% RSLogix 500 project BLUE BANNER_ORGANIC_DUMP_APR_09_2021_FAST_SLOW_BOTH_BAK083.RSS, saved by version 11.00.00.00 %
PROJECT "CCHDUMP"    % processor: MicroLogix 1400 %

PROGRAM FILES
  LAD 2   72 rungs

DATA FILES
  O0 OUTPUT  7 elements
  I1 INPUT  9 elements
  S2 STATUS  66 elements
  B3 BINARY  4 elements
  T4 TIMER  20 elements
  C5 COUNTER  1 elements
  R6 CONTROL  1 elements
  N7 INTEGER  1 elements
  F8 FLOAT  4 elements

LADDER 2
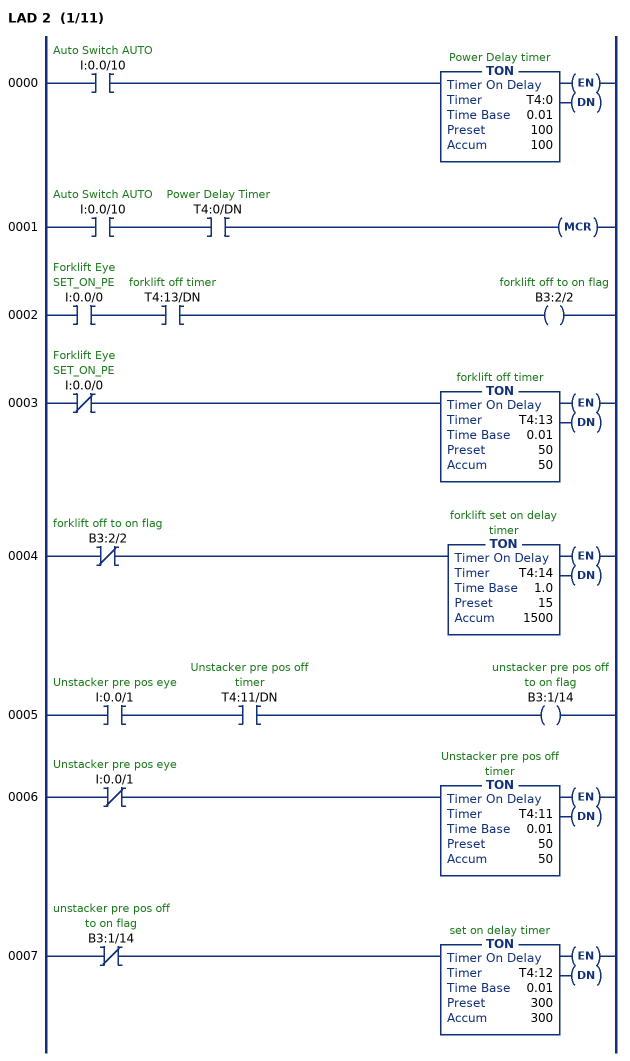
% Rung: 0 %
SOR XIC I:0.0/10 TON T4:0 0.01 100 100 EOR
%   I:0.0/10  AUTO  "Auto Switch" %
%   T4:0  "Power Delay timer" %
% Rung: 1 %
SOR XIC I:0.0/10 XIC T4:0/DN MCR EOR
%   I:0.0/10  AUTO  "Auto Switch" %
%   T4:0/DN  "Power Delay Timer" %
% Rung: 2 %
SOR XIC I:0.0/0 XIC T4:13/DN OTE B3:2/2 EOR
%   I:0.0/0  SET_ON_PE  "Forklift Eye" %
%   T4:13  "forklift off timer" %
%   B3:2/2  "forklift off to on flag" %
% Rung: 3 %
SOR XIO I:0.0/0 TON T4:13 0.01 50 50 EOR
%   I:0.0/0  SET_ON_PE  "Forklift Eye" %
%   T4:13  "forklift off timer" %
% Rung: 4 %
SOR XIO B3:2/2 TON T4:14 1.0 15 1500 EOR
%   B3:2/2  "forklift off to on flag" %
%   T4:14  "forklift set on delay timer" %
% Rung: 5 %
SOR XIC I:0.0/1 XIC T4:11/DN OTE B3:1/14 EOR
%   I:0.0/1  "Unstacker pre pos eye" %
%   T4:11  "Unstacker pre pos off timer" %
%   B3:1/14  "unstacker pre pos off to on flag" %
% Rung: 6 %
SOR XIO I:0.0/1 TON T4:11 0.01 50 50 EOR
%   I:0.0/1  "Unstacker pre pos eye" %
%   T4:11  "Unstacker pre pos off timer" %
% Rung: 7 %
SOR XIO B3:1/14 TON T4:12 0.01 300 300 EOR
%   B3:1/14  "unstacker pre pos off to on flag" %
%   T4:12  "set on delay timer" %

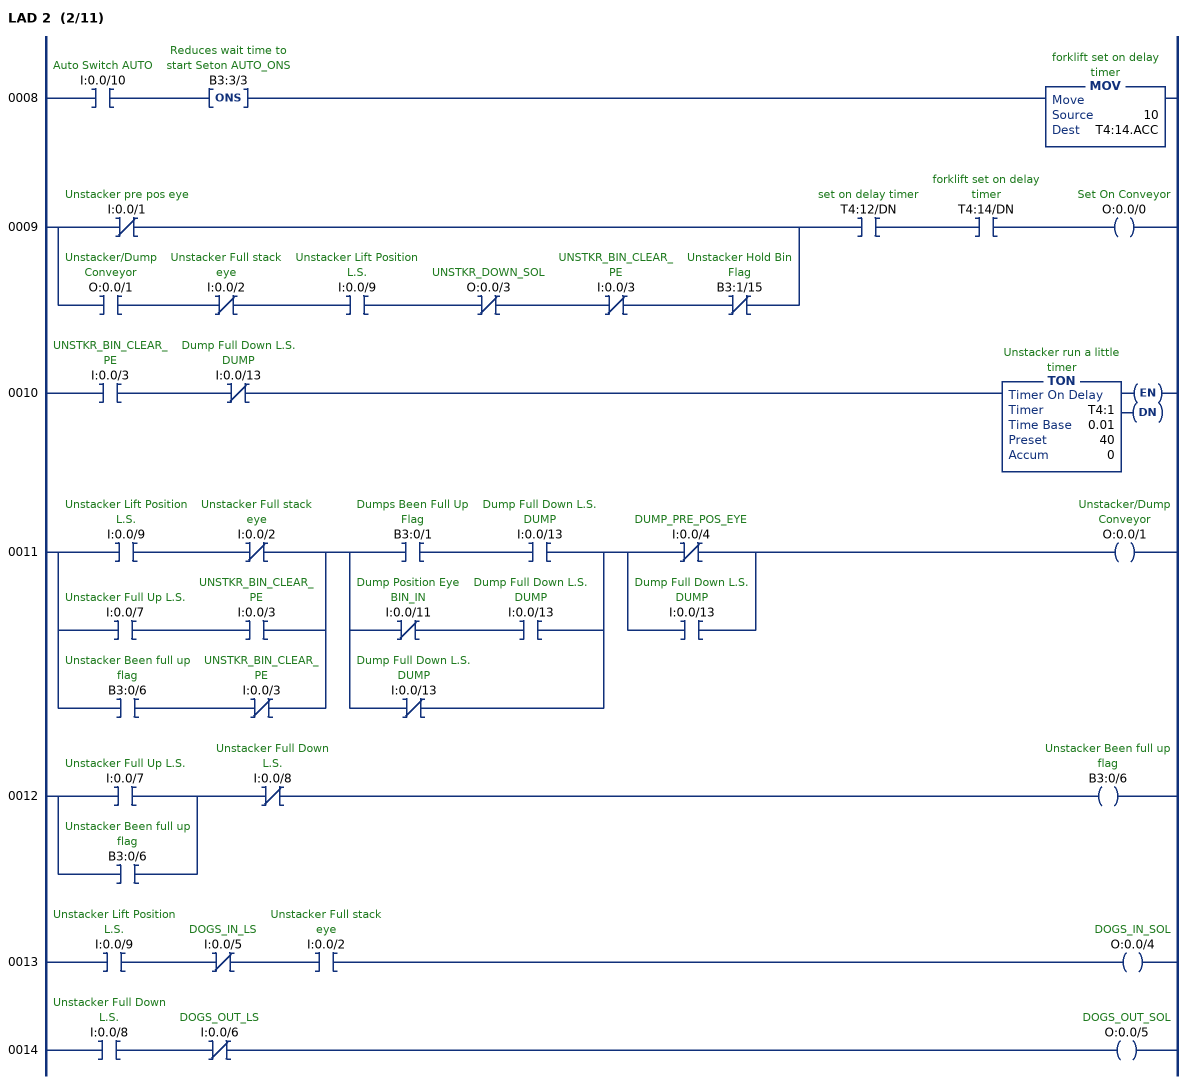
% Rung: 8 %
SOR XIC I:0.0/10 ONS B3:3/3 MOV 10 T4:14.ACC EOR
%   I:0.0/10  AUTO  "Auto Switch" %
%   B3:3/3  AUTO_ONS  "Reduces wait time to start Seton" %
%   T4:14  "forklift set on delay timer" %
% Rung: 9 %
SOR BST XIO I:0.0/1 NXB XIC O:0.0/1 XIO I:0.0/2 XIC I:0.0/9 XIO O:0.0/3 XIO I:0.0/3 XIO B3:1/15 BND XIC T4:12/DN XIC T4:14/DN OTE O:0.0/0 EOR
%   I:0.0/1  "Unstacker pre pos eye" %
%   O:0.0/1  "Unstacker/Dump Conveyor" %
%   I:0.0/2  "Unstacker Full stack eye" %
%   I:0.0/9  "Unstacker Lift Position L.S." %
%   O:0.0/3  UNSTKR_DOWN_SOL %
%   I:0.0/3  UNSTKR_BIN_CLEAR_PE %
%   B3:1/15  "Unstacker Hold Bin Flag" %
%   T4:12  "set on delay timer" %
%   T4:14  "forklift set on delay timer" %
%   O:0.0/0  "Set On Conveyor" %
% Rung: 10 %
SOR XIC I:0.0/3 XIO I:0.0/13 TON T4:1 0.01 40 0 EOR
%   I:0.0/3  UNSTKR_BIN_CLEAR_PE %
%   I:0.0/13  DUMP  "Dump Full Down L.S." %
%   T4:1  "Unstacker run a little timer" %
% Rung: 11 %
SOR BST XIC I:0.0/9 XIO I:0.0/2 NXB XIC I:0.0/7 XIC I:0.0/3 NXB XIC B3:0/6 XIO I:0.0/3 BND BST XIC B3:0/1 XIC I:0.0/13 NXB XIO I:0.0/11 XIC I:0.0/13 NXB XIO I:0.0/13 BND BST XIO I:0.0/4 NXB XIC I:0.0/13 BND OTE O:0.0/1 EOR
%   I:0.0/9  "Unstacker Lift Position L.S." %
%   I:0.0/2  "Unstacker Full stack eye" %
%   I:0.0/7  "Unstacker Full Up L.S." %
%   I:0.0/3  UNSTKR_BIN_CLEAR_PE %
%   B3:0/6  "Unstacker Been full up flag" %
%   B3:0/1  "Dumps Been Full Up Flag" %
%   I:0.0/13  DUMP  "Dump Full Down L.S." %
%   I:0.0/11  BIN_IN  "Dump Position Eye" %
%   I:0.0/4  DUMP_PRE_POS_EYE %
%   O:0.0/1  "Unstacker/Dump Conveyor" %
% Rung: 12 %
SOR BST XIC I:0.0/7 NXB XIC B3:0/6 BND XIO I:0.0/8 OTE B3:0/6 EOR
%   I:0.0/7  "Unstacker Full Up L.S." %
%   B3:0/6  "Unstacker Been full up flag" %
%   I:0.0/8  "Unstacker Full Down L.S." %
% Rung: 13 %
SOR XIC I:0.0/9 XIO I:0.0/5 XIC I:0.0/2 OTE O:0.0/4 EOR
%   I:0.0/9  "Unstacker Lift Position L.S." %
%   I:0.0/5  DOGS_IN_LS %
%   I:0.0/2  "Unstacker Full stack eye" %
%   O:0.0/4  DOGS_IN_SOL %
% Rung: 14 %
SOR XIC I:0.0/8 XIO I:0.0/6 OTE O:0.0/5 EOR
%   I:0.0/8  "Unstacker Full Down L.S." %
%   I:0.0/6  DOGS_OUT_LS %
%   O:0.0/5  DOGS_OUT_SOL %

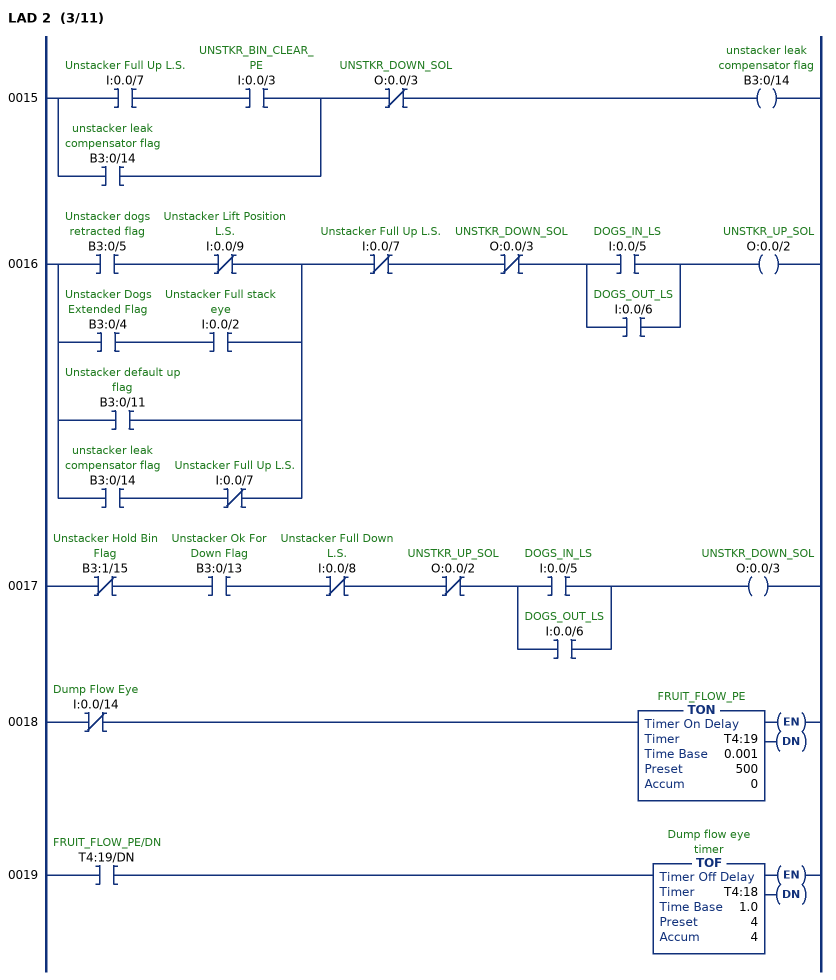
% Rung: 15 %
SOR BST XIC I:0.0/7 XIC I:0.0/3 NXB XIC B3:0/14 BND XIO O:0.0/3 OTE B3:0/14 EOR
%   I:0.0/7  "Unstacker Full Up L.S." %
%   I:0.0/3  UNSTKR_BIN_CLEAR_PE %
%   B3:0/14  "unstacker leak compensator flag" %
%   O:0.0/3  UNSTKR_DOWN_SOL %
% Rung: 16 %
SOR BST XIC B3:0/5 XIO I:0.0/9 NXB XIC B3:0/4 XIC I:0.0/2 NXB XIC B3:0/11 NXB XIC B3:0/14 XIO I:0.0/7 BND XIO I:0.0/7 XIO O:0.0/3 BST XIC I:0.0/5 NXB XIC I:0.0/6 BND OTE O:0.0/2 EOR
%   B3:0/5  "Unstacker dogs retracted flag" %
%   I:0.0/9  "Unstacker Lift Position L.S." %
%   B3:0/4  "Unstacker Dogs Extended Flag" %
%   I:0.0/2  "Unstacker Full stack eye" %
%   B3:0/11  "Unstacker default up flag" %
%   B3:0/14  "unstacker leak compensator flag" %
%   I:0.0/7  "Unstacker Full Up L.S." %
%   O:0.0/3  UNSTKR_DOWN_SOL %
%   I:0.0/5  DOGS_IN_LS %
%   I:0.0/6  DOGS_OUT_LS %
%   O:0.0/2  UNSTKR_UP_SOL %
% Rung: 17 %
SOR XIO B3:1/15 XIC B3:0/13 XIO I:0.0/8 XIO O:0.0/2 BST XIC I:0.0/5 NXB XIC I:0.0/6 BND OTE O:0.0/3 EOR
%   B3:1/15  "Unstacker Hold Bin Flag" %
%   B3:0/13  "Unstacker Ok For Down Flag" %
%   I:0.0/8  "Unstacker Full Down L.S." %
%   O:0.0/2  UNSTKR_UP_SOL %
%   I:0.0/5  DOGS_IN_LS %
%   I:0.0/6  DOGS_OUT_LS %
%   O:0.0/3  UNSTKR_DOWN_SOL %
% Rung: 18 %
SOR XIO I:0.0/14 TON T4:19 0.001 500 0 EOR
%   I:0.0/14  "Dump Flow Eye" %
%   T4:19  FRUIT_FLOW_PE %
% Rung: 19 %
SOR XIC T4:19/DN TOF T4:18 1.0 4 4 EOR
%   T4:19  FRUIT_FLOW_PE %
%   T4:18  "Dump flow eye timer" %

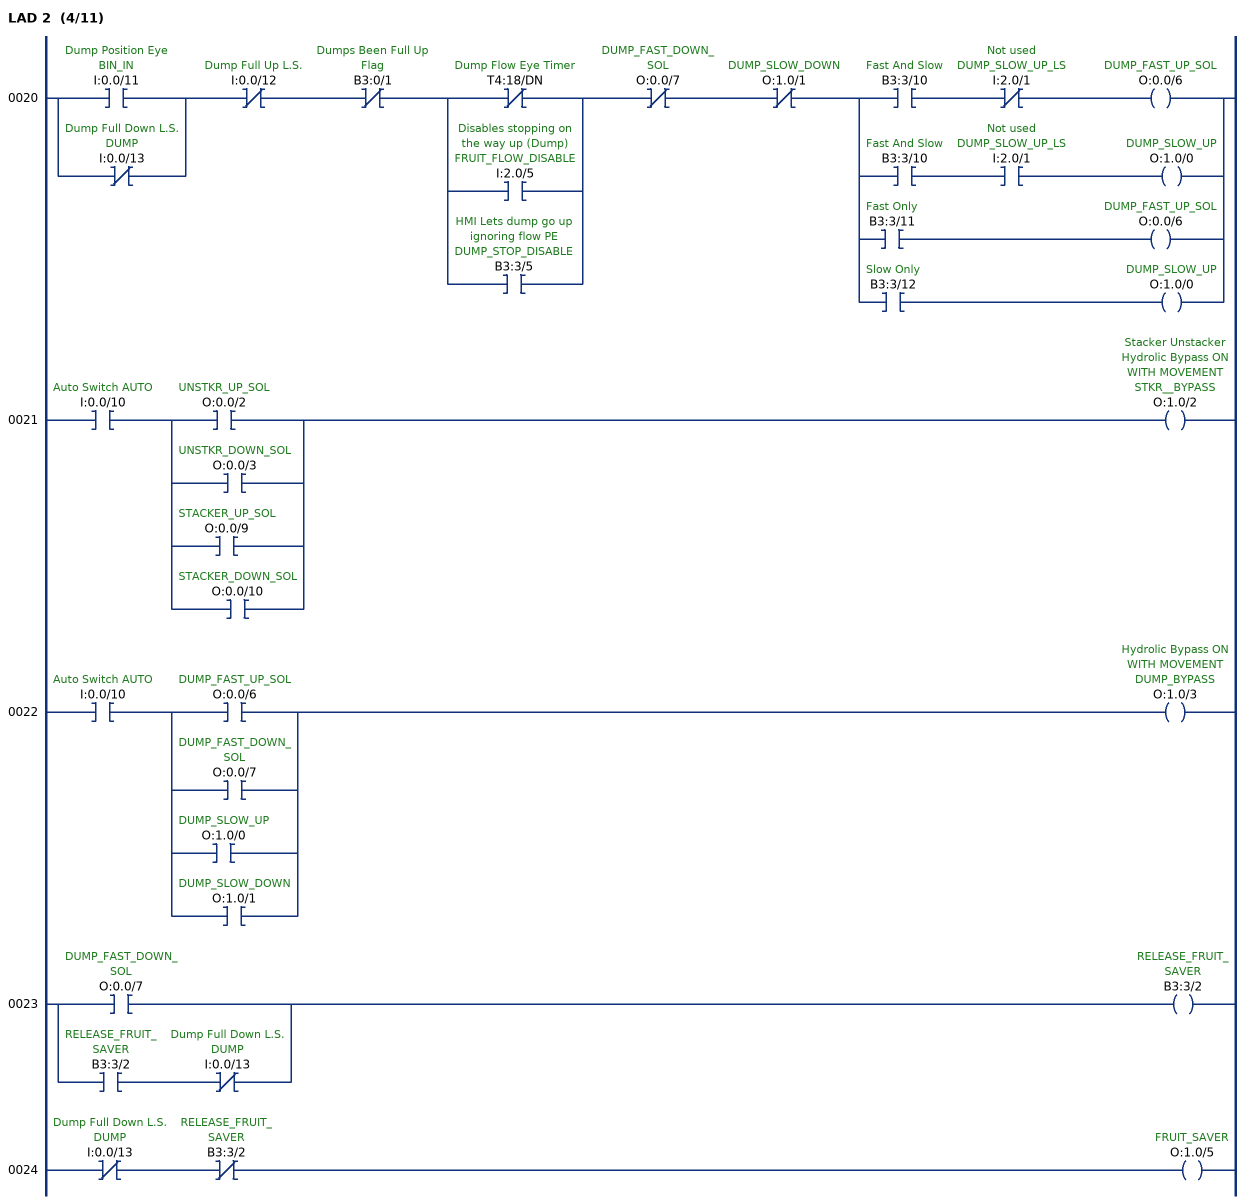
% Rung: 20 %
SOR BST XIC I:0.0/11 NXB XIO I:0.0/13 BND XIO I:0.0/12 XIO B3:0/1 BST XIO T4:18/DN NXB BST XIC I:2.0/5 NXB XIC B3:3/5 BND BND XIO O:0.0/7 XIO O:1.0/1 BST XIC B3:3/10 XIO I:2.0/1 OTE O:0.0/6 NXB XIC B3:3/10 XIC I:2.0/1 OTE O:1.0/0 NXB XIC B3:3/11 OTE O:0.0/6 NXB XIC B3:3/12 OTE O:1.0/0 BND EOR
%   I:0.0/11  BIN_IN  "Dump Position Eye" %
%   I:0.0/13  DUMP  "Dump Full Down L.S." %
%   I:0.0/12  "Dump Full Up L.S." %
%   B3:0/1  "Dumps Been Full Up Flag" %
%   T4:18/DN  "Dump Flow Eye Timer" %
%   I:2.0/5  FRUIT_FLOW_DISABLE  "Disables stopping on the way up (Dump)" %
%   B3:3/5  DUMP_STOP_DISABLE  "HMI Lets dump go up ignoring flow PE" %
%   O:0.0/7  DUMP_FAST_DOWN_SOL %
%   O:1.0/1  DUMP_SLOW_DOWN %
%   B3:3/10  "Fast And Slow" %
%   I:2.0/1  DUMP_SLOW_UP_LS  "Not used" %
%   O:0.0/6  DUMP_FAST_UP_SOL %
%   O:1.0/0  DUMP_SLOW_UP %
%   B3:3/11  "Fast Only" %
%   B3:3/12  "Slow Only" %
% Rung: 21 %
SOR XIC I:0.0/10 BST XIC O:0.0/2 NXB BST XIC O:0.0/3 NXB BST XIC O:0.0/9 NXB XIC O:0.0/10 BND BND BND OTE O:1.0/2 EOR
%   I:0.0/10  AUTO  "Auto Switch" %
%   O:0.0/2  UNSTKR_UP_SOL %
%   O:0.0/3  UNSTKR_DOWN_SOL %
%   O:0.0/9  STACKER_UP_SOL %
%   O:0.0/10  STACKER_DOWN_SOL %
%   O:1.0/2  STKR__BYPASS  "Stacker Unstacker Hydrolic Bypass ON WITH MOVEMENT" %
% Rung: 22 %
SOR XIC I:0.0/10 BST XIC O:0.0/6 NXB BST XIC O:0.0/7 NXB BST XIC O:1.0/0 NXB XIC O:1.0/1 BND BND BND OTE O:1.0/3 EOR
%   I:0.0/10  AUTO  "Auto Switch" %
%   O:0.0/6  DUMP_FAST_UP_SOL %
%   O:0.0/7  DUMP_FAST_DOWN_SOL %
%   O:1.0/0  DUMP_SLOW_UP %
%   O:1.0/1  DUMP_SLOW_DOWN %
%   O:1.0/3  DUMP_BYPASS  "Hydrolic Bypass ON WITH MOVEMENT" %
% Rung: 23 %
SOR BST XIC O:0.0/7 NXB XIC B3:3/2 XIO I:0.0/13 BND OTE B3:3/2 EOR
%   O:0.0/7  DUMP_FAST_DOWN_SOL %
%   B3:3/2  RELEASE_FRUIT_SAVER %
%   I:0.0/13  DUMP  "Dump Full Down L.S." %
% Rung: 24 %
SOR XIO I:0.0/13 XIO B3:3/2 OTE O:1.0/5 EOR
%   I:0.0/13  DUMP  "Dump Full Down L.S." %
%   B3:3/2  RELEASE_FRUIT_SAVER %
%   O:1.0/5  FRUIT_SAVER %

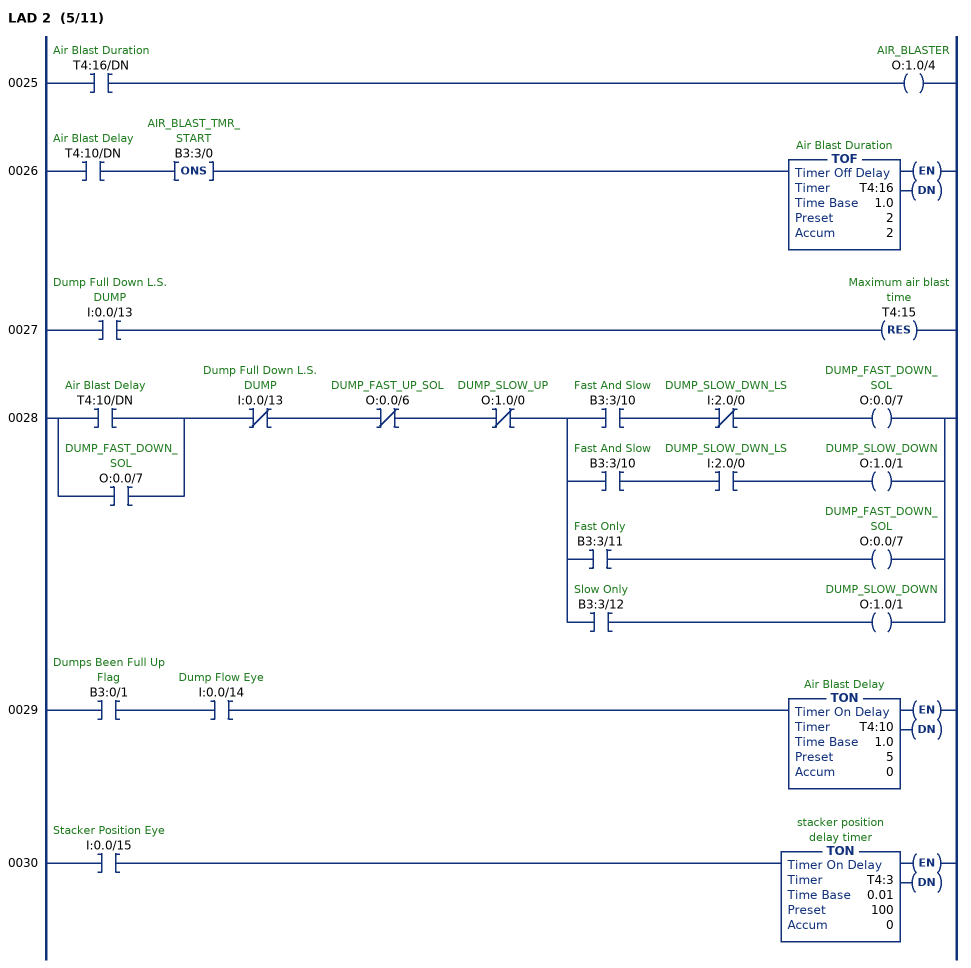
% Rung: 25 %
SOR XIC T4:16/DN OTE O:1.0/4 EOR
%   T4:16  "Air Blast Duration" %
%   O:1.0/4  AIR_BLASTER %
% Rung: 26 %
SOR XIC T4:10/DN ONS B3:3/0 TOF T4:16 1.0 2 2 EOR
%   T4:10  "Air Blast Delay" %
%   B3:3/0  AIR_BLAST_TMR_START %
%   T4:16  "Air Blast Duration" %
% Rung: 27 %
SOR XIC I:0.0/13 RES T4:15 EOR
%   I:0.0/13  DUMP  "Dump Full Down L.S." %
%   T4:15  "Maximum air blast time" %
% Rung: 28 %
SOR BST XIC T4:10/DN NXB XIC O:0.0/7 BND XIO I:0.0/13 XIO O:0.0/6 XIO O:1.0/0 BST XIC B3:3/10 XIO I:2.0/0 OTE O:0.0/7 NXB XIC B3:3/10 XIC I:2.0/0 OTE O:1.0/1 NXB XIC B3:3/11 OTE O:0.0/7 NXB XIC B3:3/12 OTE O:1.0/1 BND EOR
%   T4:10  "Air Blast Delay" %
%   O:0.0/7  DUMP_FAST_DOWN_SOL %
%   I:0.0/13  DUMP  "Dump Full Down L.S." %
%   O:0.0/6  DUMP_FAST_UP_SOL %
%   O:1.0/0  DUMP_SLOW_UP %
%   B3:3/10  "Fast And Slow" %
%   I:2.0/0  DUMP_SLOW_DWN_LS %
%   O:1.0/1  DUMP_SLOW_DOWN %
%   B3:3/11  "Fast Only" %
%   B3:3/12  "Slow Only" %
% Rung: 29 %
SOR XIC B3:0/1 XIC I:0.0/14 TON T4:10 1.0 5 0 EOR
%   B3:0/1  "Dumps Been Full Up Flag" %
%   I:0.0/14  "Dump Flow Eye" %
%   T4:10  "Air Blast Delay" %
% Rung: 30 %
SOR XIC I:0.0/15 TON T4:3 0.01 100 0 EOR
%   I:0.0/15  "Stacker Position Eye" %
%   T4:3  "stacker position delay timer" %

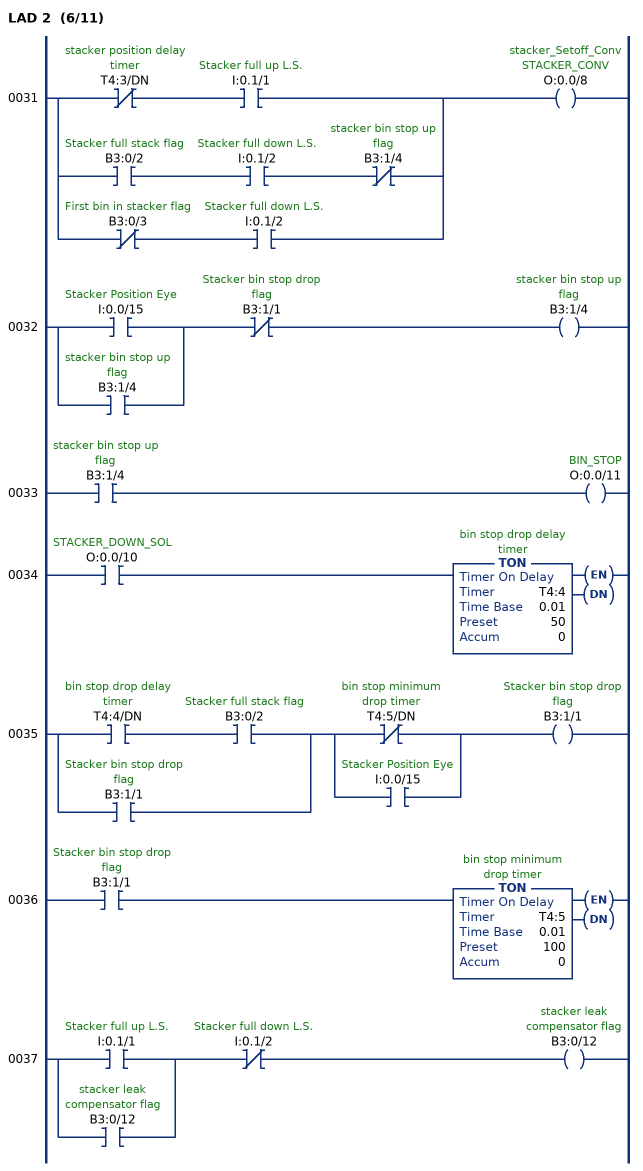
% Rung: 31 %
SOR BST XIO T4:3/DN XIC I:0.1/1 NXB XIC B3:0/2 XIC I:0.1/2 XIO B3:1/4 NXB XIO B3:0/3 XIC I:0.1/2 BND OTE O:0.0/8 EOR
%   T4:3  "stacker position delay timer" %
%   I:0.1/1  "Stacker full up L.S." %
%   B3:0/2  "Stacker full stack flag" %
%   I:0.1/2  "Stacker full down L.S." %
%   B3:1/4  "stacker bin stop up flag" %
%   B3:0/3  "First bin in stacker flag" %
%   O:0.0/8  STACKER_CONV  "stacker_Setoff_Conv" %
% Rung: 32 %
SOR BST XIC I:0.0/15 NXB XIC B3:1/4 BND XIO B3:1/1 OTE B3:1/4 EOR
%   I:0.0/15  "Stacker Position Eye" %
%   B3:1/4  "stacker bin stop up flag" %
%   B3:1/1  "Stacker bin stop drop flag" %
% Rung: 33 %
SOR XIC B3:1/4 OTE O:0.0/11 EOR
%   B3:1/4  "stacker bin stop up flag" %
%   O:0.0/11  BIN_STOP %
% Rung: 34 %
SOR XIC O:0.0/10 TON T4:4 0.01 50 0 EOR
%   O:0.0/10  STACKER_DOWN_SOL %
%   T4:4  "bin stop drop delay timer" %
% Rung: 35 %
SOR BST XIC T4:4/DN XIC B3:0/2 NXB XIC B3:1/1 BND BST XIO T4:5/DN NXB XIC I:0.0/15 BND OTE B3:1/1 EOR
%   T4:4  "bin stop drop delay timer" %
%   B3:0/2  "Stacker full stack flag" %
%   B3:1/1  "Stacker bin stop drop flag" %
%   T4:5  "bin stop minimum drop timer" %
%   I:0.0/15  "Stacker Position Eye" %
% Rung: 36 %
SOR XIC B3:1/1 TON T4:5 0.01 100 0 EOR
%   B3:1/1  "Stacker bin stop drop flag" %
%   T4:5  "bin stop minimum drop timer" %
% Rung: 37 %
SOR BST XIC I:0.1/1 NXB XIC B3:0/12 BND XIO I:0.1/2 OTE B3:0/12 EOR
%   I:0.1/1  "Stacker full up L.S." %
%   B3:0/12  "stacker leak compensator flag" %
%   I:0.1/2  "Stacker full down L.S." %

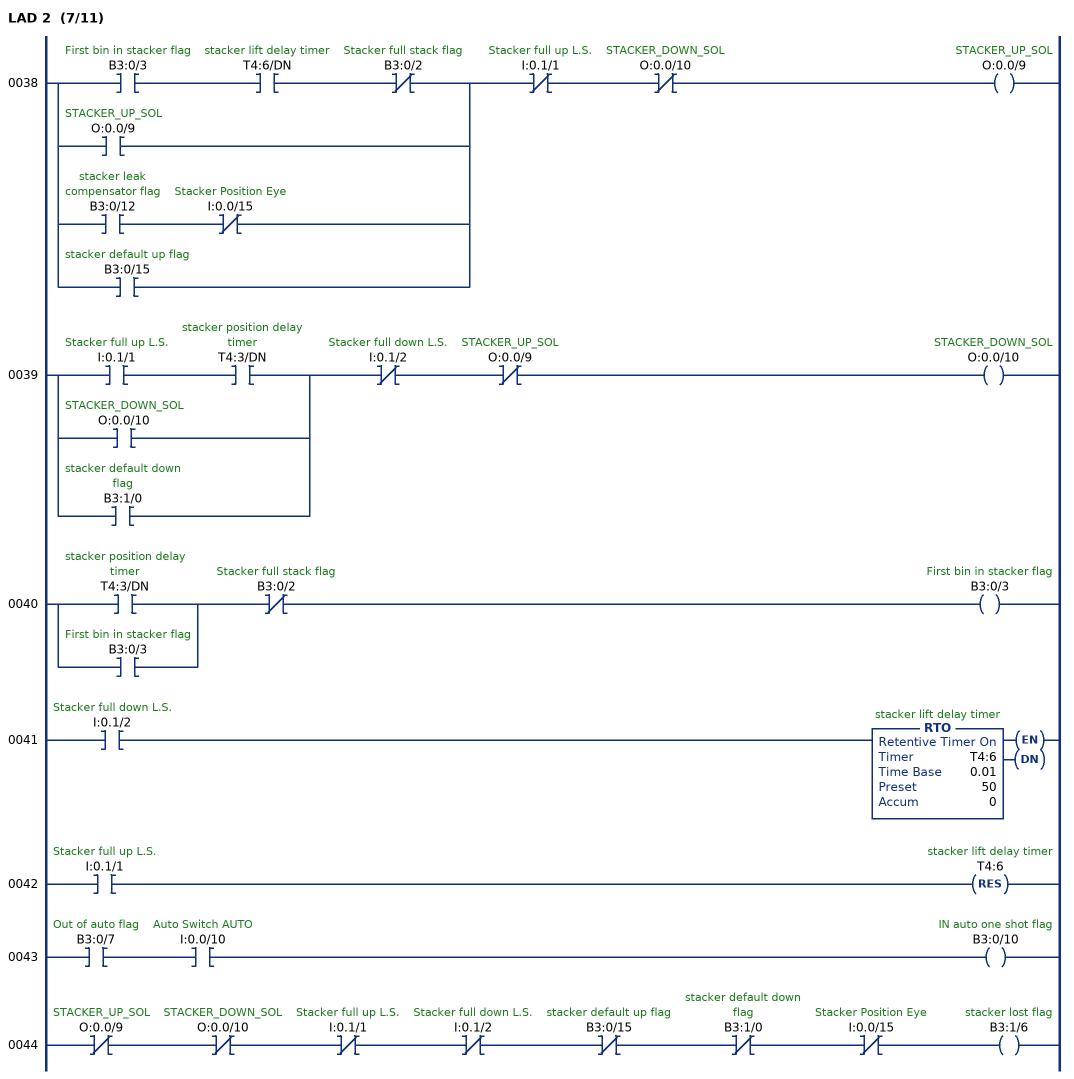
% Rung: 38 %
SOR BST XIC B3:0/3 XIC T4:6/DN XIO B3:0/2 NXB XIC O:0.0/9 NXB XIC B3:0/12 XIO I:0.0/15 NXB XIC B3:0/15 BND XIO I:0.1/1 XIO O:0.0/10 OTE O:0.0/9 EOR
%   B3:0/3  "First bin in stacker flag" %
%   T4:6  "stacker lift delay timer" %
%   B3:0/2  "Stacker full stack flag" %
%   O:0.0/9  STACKER_UP_SOL %
%   B3:0/12  "stacker leak compensator flag" %
%   I:0.0/15  "Stacker Position Eye" %
%   B3:0/15  "stacker default up flag" %
%   I:0.1/1  "Stacker full up L.S." %
%   O:0.0/10  STACKER_DOWN_SOL %
% Rung: 39 %
SOR BST XIC I:0.1/1 XIC T4:3/DN NXB XIC O:0.0/10 NXB XIC B3:1/0 BND XIO I:0.1/2 XIO O:0.0/9 OTE O:0.0/10 EOR
%   I:0.1/1  "Stacker full up L.S." %
%   T4:3  "stacker position delay timer" %
%   O:0.0/10  STACKER_DOWN_SOL %
%   B3:1/0  "stacker default down flag" %
%   I:0.1/2  "Stacker full down L.S." %
%   O:0.0/9  STACKER_UP_SOL %
% Rung: 40 %
SOR BST XIC T4:3/DN NXB XIC B3:0/3 BND XIO B3:0/2 OTE B3:0/3 EOR
%   T4:3  "stacker position delay timer" %
%   B3:0/3  "First bin in stacker flag" %
%   B3:0/2  "Stacker full stack flag" %
% Rung: 41 %
SOR XIC I:0.1/2 RTO T4:6 0.01 50 0 EOR
%   I:0.1/2  "Stacker full down L.S." %
%   T4:6  "stacker lift delay timer" %
% Rung: 42 %
SOR XIC I:0.1/1 RES T4:6 EOR
%   I:0.1/1  "Stacker full up L.S." %
%   T4:6  "stacker lift delay timer" %
% Rung: 43 %
SOR XIC B3:0/7 XIC I:0.0/10 OTE B3:0/10 EOR
%   B3:0/7  "Out of auto flag" %
%   I:0.0/10  AUTO  "Auto Switch" %
%   B3:0/10  "IN auto one shot flag" %
% Rung: 44 %
SOR XIO O:0.0/9 XIO O:0.0/10 XIO I:0.1/1 XIO I:0.1/2 XIO B3:0/15 XIO B3:1/0 XIO I:0.0/15 OTE B3:1/6 EOR
%   O:0.0/9  STACKER_UP_SOL %
%   O:0.0/10  STACKER_DOWN_SOL %
%   I:0.1/1  "Stacker full up L.S." %
%   I:0.1/2  "Stacker full down L.S." %
%   B3:0/15  "stacker default up flag" %
%   B3:1/0  "stacker default down flag" %
%   I:0.0/15  "Stacker Position Eye" %
%   B3:1/6  "stacker lost flag" %

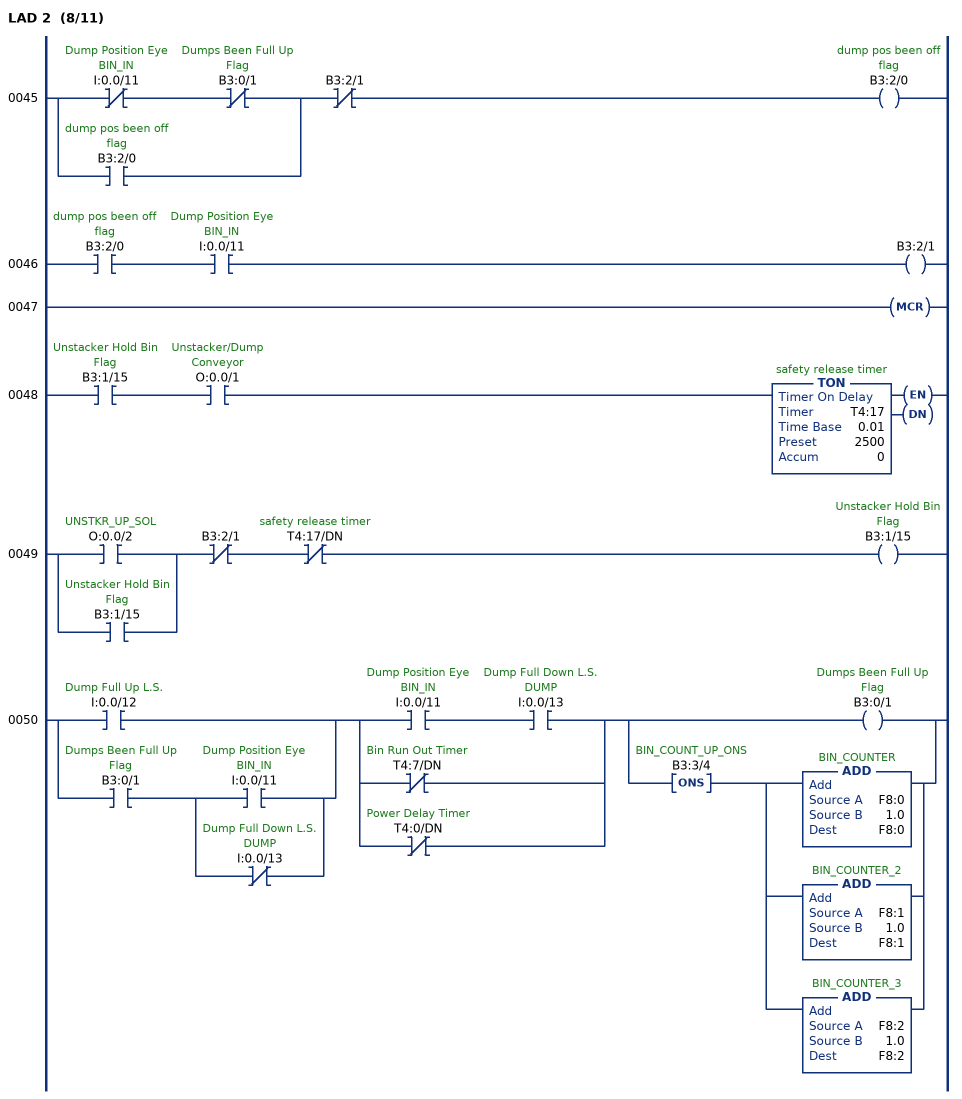
% Rung: 45 %
SOR BST XIO I:0.0/11 XIO B3:0/1 NXB XIC B3:2/0 BND XIO B3:2/1 OTE B3:2/0 EOR
%   I:0.0/11  BIN_IN  "Dump Position Eye" %
%   B3:0/1  "Dumps Been Full Up Flag" %
%   B3:2/0  "dump pos been off flag" %
% Rung: 46 %
SOR XIC B3:2/0 XIC I:0.0/11 OTE B3:2/1 EOR
%   B3:2/0  "dump pos been off flag" %
%   I:0.0/11  BIN_IN  "Dump Position Eye" %
% Rung: 47 %
SOR MCR EOR
% Rung: 48 %
SOR XIC B3:1/15 XIC O:0.0/1 TON T4:17 0.01 2500 0 EOR
%   B3:1/15  "Unstacker Hold Bin Flag" %
%   O:0.0/1  "Unstacker/Dump Conveyor" %
%   T4:17  "safety release timer" %
% Rung: 49 %
SOR BST XIC O:0.0/2 NXB XIC B3:1/15 BND XIO B3:2/1 XIO T4:17/DN OTE B3:1/15 EOR
%   O:0.0/2  UNSTKR_UP_SOL %
%   B3:1/15  "Unstacker Hold Bin Flag" %
%   T4:17  "safety release timer" %
% Rung: 50 %
SOR BST XIC I:0.0/12 NXB XIC B3:0/1 BST XIC I:0.0/11 NXB XIO I:0.0/13 BND BND BST XIC I:0.0/11 XIC I:0.0/13 NXB XIO T4:7/DN NXB XIO T4:0/DN BND BST OTE B3:0/1 NXB ONS B3:3/4 BST ADD F8:0 1.0 F8:0 NXB BST ADD F8:1 1.0 F8:1 NXB ADD F8:2 1.0 F8:2 BND BND BND EOR
%   I:0.0/12  "Dump Full Up L.S." %
%   B3:0/1  "Dumps Been Full Up Flag" %
%   I:0.0/11  BIN_IN  "Dump Position Eye" %
%   I:0.0/13  DUMP  "Dump Full Down L.S." %
%   T4:7/DN  "Bin Run Out Timer" %
%   T4:0/DN  "Power Delay Timer" %
%   B3:3/4  BIN_COUNT_UP_ONS %
%   F8:0  BIN_COUNTER %
%   F8:1  BIN_COUNTER_2 %
%   F8:2  BIN_COUNTER_3 %

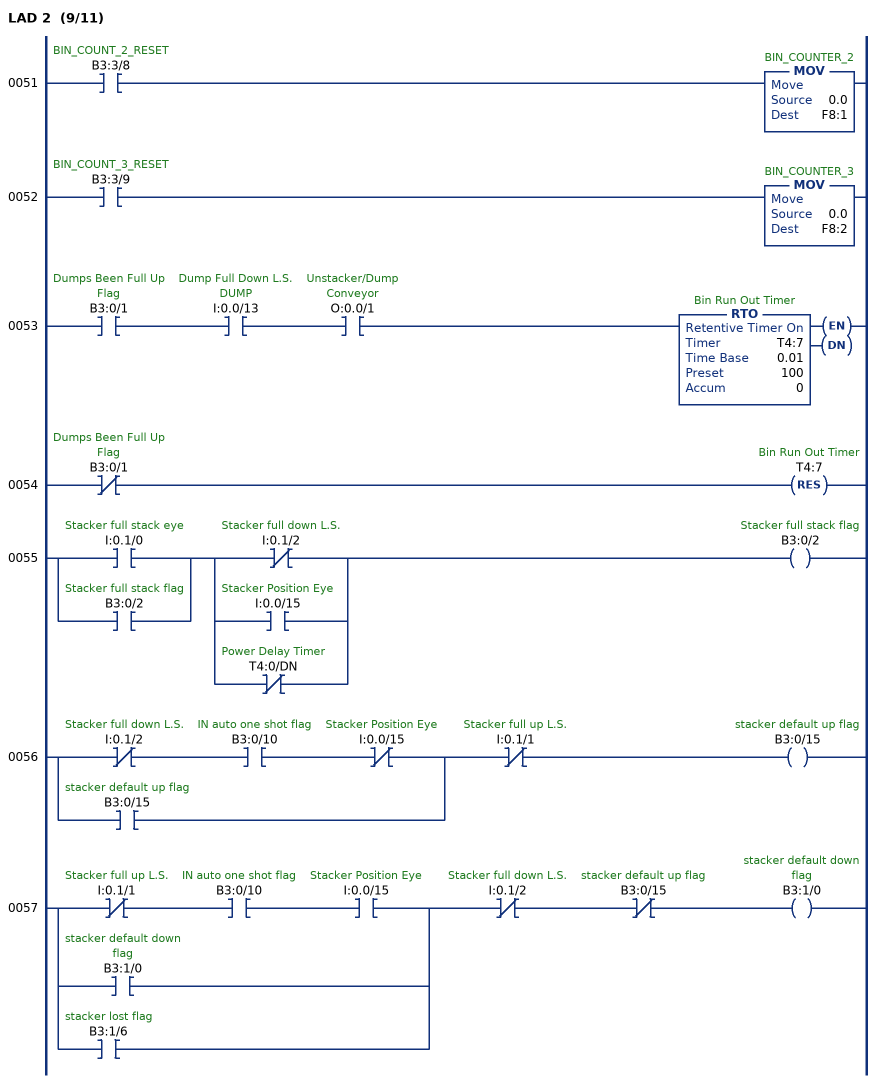
% Rung: 51 %
SOR XIC B3:3/8 MOV 0.0 F8:1 EOR
%   B3:3/8  BIN_COUNT_2_RESET %
%   F8:1  BIN_COUNTER_2 %
% Rung: 52 %
SOR XIC B3:3/9 MOV 0.0 F8:2 EOR
%   B3:3/9  BIN_COUNT_3_RESET %
%   F8:2  BIN_COUNTER_3 %
% Rung: 53 %
SOR XIC B3:0/1 XIC I:0.0/13 XIC O:0.0/1 RTO T4:7 0.01 100 0 EOR
%   B3:0/1  "Dumps Been Full Up Flag" %
%   I:0.0/13  DUMP  "Dump Full Down L.S." %
%   O:0.0/1  "Unstacker/Dump Conveyor" %
%   T4:7  "Bin Run Out Timer" %
% Rung: 54 %
SOR XIO B3:0/1 RES T4:7 EOR
%   B3:0/1  "Dumps Been Full Up Flag" %
%   T4:7  "Bin Run Out Timer" %
% Rung: 55 %
SOR BST XIC I:0.1/0 NXB XIC B3:0/2 BND BST XIO I:0.1/2 NXB XIC I:0.0/15 NXB XIO T4:0/DN BND OTE B3:0/2 EOR
%   I:0.1/0  "Stacker full stack eye" %
%   B3:0/2  "Stacker full stack flag" %
%   I:0.1/2  "Stacker full down L.S." %
%   I:0.0/15  "Stacker Position Eye" %
%   T4:0/DN  "Power Delay Timer" %
% Rung: 56 %
SOR BST XIO I:0.1/2 XIC B3:0/10 XIO I:0.0/15 NXB XIC B3:0/15 BND XIO I:0.1/1 OTE B3:0/15 EOR
%   I:0.1/2  "Stacker full down L.S." %
%   B3:0/10  "IN auto one shot flag" %
%   I:0.0/15  "Stacker Position Eye" %
%   B3:0/15  "stacker default up flag" %
%   I:0.1/1  "Stacker full up L.S." %
% Rung: 57 %
SOR BST XIO I:0.1/1 XIC B3:0/10 XIC I:0.0/15 NXB XIC B3:1/0 NXB XIC B3:1/6 BND XIO I:0.1/2 XIO B3:0/15 OTE B3:1/0 EOR
%   I:0.1/1  "Stacker full up L.S." %
%   B3:0/10  "IN auto one shot flag" %
%   I:0.0/15  "Stacker Position Eye" %
%   B3:1/0  "stacker default down flag" %
%   B3:1/6  "stacker lost flag" %
%   I:0.1/2  "Stacker full down L.S." %
%   B3:0/15  "stacker default up flag" %

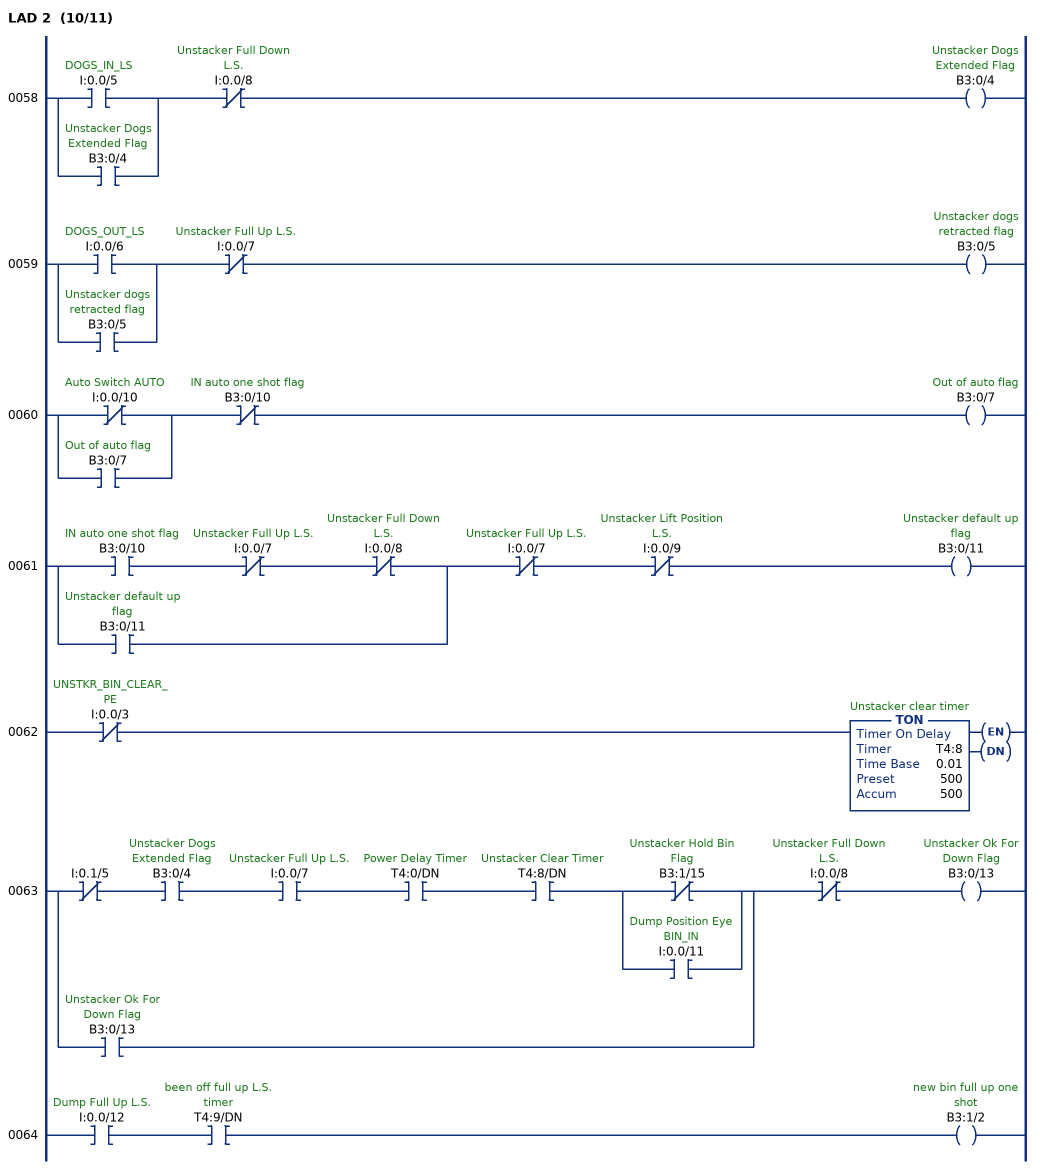
% Rung: 58 %
SOR BST XIC I:0.0/5 NXB XIC B3:0/4 BND XIO I:0.0/8 OTE B3:0/4 EOR
%   I:0.0/5  DOGS_IN_LS %
%   B3:0/4  "Unstacker Dogs Extended Flag" %
%   I:0.0/8  "Unstacker Full Down L.S." %
% Rung: 59 %
SOR BST XIC I:0.0/6 NXB XIC B3:0/5 BND XIO I:0.0/7 OTE B3:0/5 EOR
%   I:0.0/6  DOGS_OUT_LS %
%   B3:0/5  "Unstacker dogs retracted flag" %
%   I:0.0/7  "Unstacker Full Up L.S." %
% Rung: 60 %
SOR BST XIO I:0.0/10 NXB XIC B3:0/7 BND XIO B3:0/10 OTE B3:0/7 EOR
%   I:0.0/10  AUTO  "Auto Switch" %
%   B3:0/7  "Out of auto flag" %
%   B3:0/10  "IN auto one shot flag" %
% Rung: 61 %
SOR BST XIC B3:0/10 XIO I:0.0/7 XIO I:0.0/8 NXB XIC B3:0/11 BND XIO I:0.0/7 XIO I:0.0/9 OTE B3:0/11 EOR
%   B3:0/10  "IN auto one shot flag" %
%   I:0.0/7  "Unstacker Full Up L.S." %
%   I:0.0/8  "Unstacker Full Down L.S." %
%   B3:0/11  "Unstacker default up flag" %
%   I:0.0/9  "Unstacker Lift Position L.S." %
% Rung: 62 %
SOR XIO I:0.0/3 TON T4:8 0.01 500 500 EOR
%   I:0.0/3  UNSTKR_BIN_CLEAR_PE %
%   T4:8  "Unstacker clear timer" %
% Rung: 63 %
SOR BST XIO I:0.1/5 XIC B3:0/4 XIC I:0.0/7 XIC T4:0/DN XIC T4:8/DN BST XIO B3:1/15 NXB XIC I:0.0/11 BND NXB XIC B3:0/13 BND XIO I:0.0/8 OTE B3:0/13 EOR
%   B3:0/4  "Unstacker Dogs Extended Flag" %
%   I:0.0/7  "Unstacker Full Up L.S." %
%   T4:0/DN  "Power Delay Timer" %
%   T4:8/DN  "Unstacker Clear Timer" %
%   B3:1/15  "Unstacker Hold Bin Flag" %
%   I:0.0/11  BIN_IN  "Dump Position Eye" %
%   B3:0/13  "Unstacker Ok For Down Flag" %
%   I:0.0/8  "Unstacker Full Down L.S." %
% Rung: 64 %
SOR XIC I:0.0/12 XIC T4:9/DN OTE B3:1/2 EOR
%   I:0.0/12  "Dump Full Up L.S." %
%   T4:9  "been off full up L.S. timer" %
%   B3:1/2  "new bin full up one shot" %

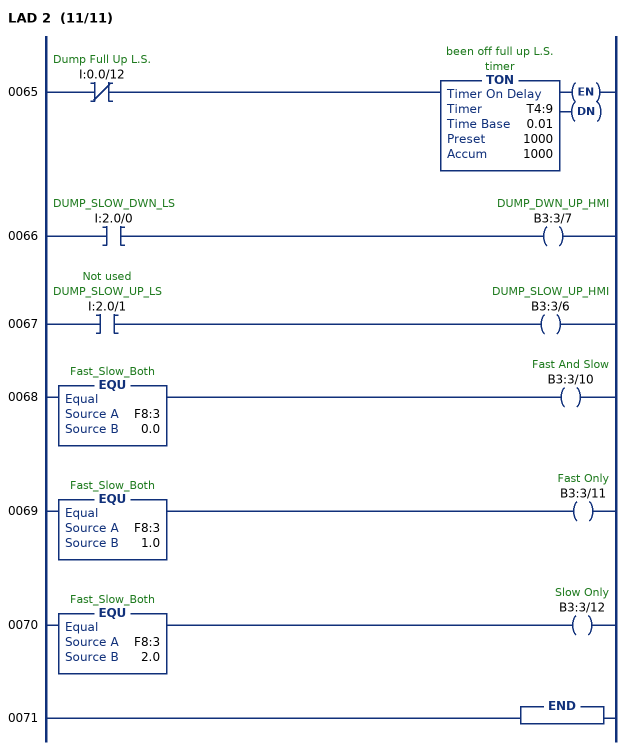
% Rung: 65 %
SOR XIO I:0.0/12 TON T4:9 0.01 1000 1000 EOR
%   I:0.0/12  "Dump Full Up L.S." %
%   T4:9  "been off full up L.S. timer" %
% Rung: 66 %
SOR XIC I:2.0/0 OTE B3:3/7 EOR
%   I:2.0/0  DUMP_SLOW_DWN_LS %
%   B3:3/7  DUMP_DWN_UP_HMI %
% Rung: 67 %
SOR XIC I:2.0/1 OTE B3:3/6 EOR
%   I:2.0/1  DUMP_SLOW_UP_LS  "Not used" %
%   B3:3/6  DUMP_SLOW_UP_HMI %
% Rung: 68 %
SOR EQU F8:3 0.0 OTE B3:3/10 EOR
%   F8:3  "Fast_Slow_Both" %
%   B3:3/10  "Fast And Slow" %
% Rung: 69 %
SOR EQU F8:3 1.0 OTE B3:3/11 EOR
%   F8:3  "Fast_Slow_Both" %
%   B3:3/11  "Fast Only" %
% Rung: 70 %
SOR EQU F8:3 2.0 OTE B3:3/12 EOR
%   F8:3  "Fast_Slow_Both" %
%   B3:3/12  "Slow Only" %
% Rung: 71 %
SOR END EOR

OTHER DOCUMENTED ADDRESSES
  B3:3/1  NOT_USED
  I:2.0/2  UNSTK_DOGS_OUT
  I:2.0/3  UNSTKR_DOGS_OUT2  "Not Used"
  N7:0  SET_ON_TIMER  "HMI"
  O:0.0/12  AIR_BLAST  "Bin dump air blast solenoid"
  T4:2  SLOW_DELAY_OFF  "Bin in off delay"
  T4:2/DN  SLO  "Dump Flow Clear Timer"

REVISION NOTES
  0: Eidenburg Bin Dump
  2: Extra Counters
  3: new limit switch
  4: interlock added apr 5 2021

DATA TABLE (non-zero values as saved)
DATA B3
% B3:0 % 0X00A0 0X8000 0X0000 0X00A0
DATA T4
% .PRE .ACC %
% T4:0 % 100 100
% T4:1 % 40 0
% T4:2 % 4 2
% T4:3 % 100 0
% T4:4 % 50 0
% T4:5 % 100 0
% T4:6 % 50 0
% T4:7 % 100 0
% T4:8 % 500 500
% T4:9 % 1000 1000
% T4:10 % 5 0
% T4:11 % 50 50
% T4:12 % 300 300
% T4:13 % 50 50
% T4:14 % 15 1500
% T4:15 % 500 0
% T4:16 % 2 2
% T4:17 % 2500 0
% T4:18 % 4 4
% T4:19 % 500 0
DATA F8
% F8:0 % 2 0 0 0
